TYPE stInfoData :
STRUCT
	State 		AT %I* : WORD;
	InfoData 	AT %I* : AMSADDR;
END_STRUCT
END_TYPE

(* stored: Version 1.1.0.1, ProductVersion 3.1.4022.6
   DUT stInfoData: Id {b6a6ce2d-e3fc-4743-987b-cde97d1a7d4e} *)
